{attribute 'GeneratedUsingTerminal: EK1122-0000-0018'}
{attribute addProperty BoxType "EK1122-0000-0018"}
{attribute addProperty Id "Beckhoff_EKxxxx_0080sub_EK1100EK1100_1FC0878B2"}
{attribute addProperty CRC "2629449202"}
{attribute addProperty Size "2"}
TYPE Beckhoff_EKxxxx_0080EK1122_9CBA35F2 EXTENDS EK1122_1FC0878B :
STRUCT
	{attribute addProperty Name "Beckhoff_EKxxxx_0080sub_EK1100"}
	{attribute addProperty PreviousPort "Beckhoff EKxxxx-0080EK1122 : D"}
	Beckhoff_EKxxxx_0080sub_EK1100 : EK1100_1FC0878B;
END_STRUCT
END_TYPE

(* stored: Version 1.2.0.0, ProductVersion 3.1.4024.9
   DUT Beckhoff_EKxxxx_0080EK1122_9CBA35F2: Id {bef6c50d-5bc0-4c18-91ad-e5d9136b6fa2} *)
